// TIA Portal V19 export
TYPE "LPMLV2022_typeDiagnostics"
TITLE = LPMLV2022_typeDiagnostics
// Support: tech.team.motioncontrol@siemens.com
// stored: Access Published
   STRUCT
      bufferIndex { ExternalWritable := 'False'} : Int := -1;   // Index of actual buffer entry
      buffer { ExternalWritable := 'False'} : Array[0.."LPMLV2022_DIAG_BUFFER_UPPER_LIM"] of "LPMLV2022_typeDiagnosticsEntry";   // Diagnostics information buffer
   END_STRUCT;
END_TYPE
